FUNCTION F_LogContext : I_ContextBuilder
VAR_INPUT
END_VAR
VAR
END_VAR

END_FUNCTION

(* stored: Version 1.1.0.1, ProductVersion 3.1.4024.0
   POU F_LogContext: Id {15bc0808-4d58-45ab-93cf-1a8d645eec0b}, SpecialFunc None *)
